FUNCTION_BLOCK Conveyor
VAR_INPUT
	bEnable : BOOL;
END_VAR
VAR_OUTPUT	
	enable AT %Q* : BOOL;
	direction AT %Q* : BOOL; //FALSE = forward, TRUE = backward
	pulse AT %Q* : BOOL;
	reset AT %Q* : BOOL;
	
	error AT %I* : BOOL;
	sensorEntry AT %I* : BOOL;
	sensorExit AT %I* : BOOL;
	
	//vertical conveyors only
	requestLifter: BOOL;

	lifterEnable AT %Q* : BOOL := TRUE;
	lifterDirection AT %Q* : BOOL; //FALSE = up, TRUE = down
	lifterPulse AT %Q* : BOOL;
	lifterReset AT %Q* : BOOL;
	
	lifterError AT %I* : BOOL;
	extended AT %I* : BOOL;
	retracted AT %I* : BOOL;
END_VAR
VAR_OUTPUT
	position AT %I* : REAL;
	velocity AT %I* : REAL;
END_VAR
VAR
	operation : ConveyorMode;
	request : ConveyorMode;
	
	//pulses are assumed to be low-HIGH-low
	pulser : TP;
	lifterPulser : TP;
	
	hasLifter : BOOL;
END_VAR
VAR_STAT CONSTANT
	pulseWidth : TIME := T#25MS;
END_VAR

pulser(IN:= , PT:= pulseWidth, Q=> pulse, ET=> );

direction := (operation = ConveyorMode.BACKWARD);

pulser.IN := 
	enable AND 
	NOT error AND 
	NOT reset AND 
	(operation = ConveyorMode.FORWARD OR operation = ConveyorMode.BACKWARD);

IF pulser.IN AND NOT pulser.Q THEN
	pulser.IN := FALSE;
END_IF

lifterPulser(IN:= , PT:= pulseWidth, Q=> lifterPulse, ET=> );

lifterPulser.IN := 
	hasLifter AND
	lifterEnable AND 
	NOT lifterError AND 
	NOT lifterReset AND 
	requestLifter;
	
IF lifterPulser.IN AND NOT lifterPulser.Q THEN
	lifterPulser.IN := FALSE;
END_IF

METHOD backward : BOOL
VAR_INPUT
END_VAR
END_METHOD

METHOD extend : BOOL
VAR_INPUT
END_VAR
END_METHOD

METHOD forward : BOOL
VAR_INPUT
END_VAR
END_METHOD

METHOD occupied : BOOL
occupied := sensorExit OR sensorEntry;
END_METHOD

METHOD reset : BOOL
VAR_INPUT
END_VAR
position := 0;
velocity := velocity; //no change

extend();
END_METHOD

METHOD retract : BOOL
VAR_INPUT
END_VAR
END_METHOD

METHOD setOperation : BOOL
VAR_INPUT
	newOperation : ConveyorMode;
END_VAR
operation := newOperation;
END_METHOD

METHOD setRequest : BOOL
VAR_INPUT
	requestedMode : ConveyorMode;
END_VAR
request := requestedMode;
END_METHOD

METHOD target : BOOL
VAR_INPUT
	targetPosition : REAL;
END_VAR
END_METHOD

END_FUNCTION_BLOCK

(* stored: Version 1.1.0.1, ProductVersion 3.1.4024.11
   POU Conveyor: Id {de162f93-5907-4a07-a0b5-f0d4a4560d6a}, SpecialFunc None
   Method backward: Id {86f9a8ba-67b5-4107-b253-01b957c1bf10}
   Method extend: Id {8f868bfa-a538-4183-8601-28b224890cc0}
   Method forward: Id {87d44885-25ee-41d2-af0e-9e2311376d2b}
   Method occupied: Id {1a437e43-b177-4373-bb48-3c058bcf1a3f}
   Method reset: Id {d40da114-e5c3-466f-8119-1749f88356bf}
   Method retract: Id {e67cd767-48c0-4514-8169-49f3436776ec}
   Method setOperation: Id {0ffca73b-6343-4082-96ff-fb3a381bc240}
   Method setRequest: Id {c2bcb45d-32a3-4c3d-ac25-48dd409d79ec}
   Method target: Id {ea17b475-eaf3-4273-b8f8-a97119ee998d} *)
